# B&R Automation Studio project Nitto (part 18)

#### picctrl.ab
```automation-basic
PROGRAM _INIT
(* init program *)
wPageAct := wPageAct;
wPageOld := 255;
//wPageNew := wPageNew;
// 2012-09-11 /schoenefeldr/
wPageNew := 2;
wPageNo  := 255;

wLanguageAct := wLanguageAct;
wLanguageNew := wLanguageNew;

//-------------------------------
//access to local structures
strcpy(ADR(szPvName), "csv_hdl:CSV_Hndl");
wStatus := PV_xgetadr(ADR(szPvName),ADR(lAdrCSV_Hndl),ADR(lDataLen));
IF (wStatus = 0) THEN
	ptCSV_Hndl ACCESS lAdrCSV_Hndl;
ENDIF;

strcpy(ADR(szPvName), "tool_hdl:TOOL_Hndl");
wStatus := PV_xgetadr(ADR(szPvName),ADR(lAdrTool_Hndl),ADR(lDataLen));
IF (wStatus = 0) THEN
	ptTool_Hndl ACCESS lAdrTool_Hndl;
ENDIF;

strcpy(ADR(szPvName), "save2USB:BackupRecipes2USB");
wStatus := PV_xgetadr(ADR(szPvName),ADR(lAdrBackupRecipes2USB),ADR(lDataLen));
IF (wStatus = 0) THEN
	ptBackupRecipes2USB ACCESS lAdrBackupRecipes2USB;
ENDIF;

strcpy(ADR(szPvName), "save2USB:BackupTools2USB");
wStatus := PV_xgetadr(ADR(szPvName),ADR(lAdrBackupTools2USB),ADR(lDataLen));
IF (wStatus = 0) THEN
	ptBackupTools2USB ACCESS lAdrBackupTools2USB;
ENDIF;

strcpy(ADR(szPvName), "tool_hdl:szFileDevice");
wStatus := PV_xgetadr(ADR(szPvName),ADR(lAdrFileDeviceTool),ADR(lDataLen));
IF (wStatus = 0) THEN
	ptFileDeviceTool ACCESS lAdrFileDeviceTool;
ENDIF;

strcpy(ADR(szPvName), "tool_hdl:tmpTool");
wStatus := PV_xgetadr(ADR(szPvName),ADR(lAdrTmpTool),ADR(lDataLen));
IF (wStatus = 0) THEN
	ptTmpTool ACCESS lAdrTmpTool;
ENDIF;

	HWInfo_0.enable := TRUE;
	HWInfo_0.first := TRUE;
	HWInfo_0.pName := ADR(HWString);
	HWInfo_0 FUB HWInfo();

	AssignFirstListboxIdx		:= TRUE;
	FirstListboxIdxValid		:= FALSE;

END_PROGRAM

PROGRAM _CYCLIC
(* cyclic program *)
	TON_Cal.IN	:= (gVisu.Cmd.pageSel.actPage = 100)
	TON_Cal.PT	:= T#10s
	TON_Cal FUB TON();

	strcpy(ADR(HWString), "AR000");	//OKrebs 17.06.2014

	IF (HWString = "AR000") THEN
		IF (gVisu.Cmd.pageSel.actPage = 100) THEN
			gVisu.Cmd.pageSel.newPage := 2;
		ENDIF
	ELSE
		IF (CalibrationState = 1) AND (TON_Cal.Q) THEN
			gVisu.Cmd.pageSel.newPage := 2;
		ENDIF;
	ENDIF;

	wPageAct:=	gVisu.Cmd.pageSel.actPage

	;Blinker
TP_10ms_01.IN := NOT (TP_10ms_02.Q);
TP_10ms_01 FUB TP_10ms();
TP_10ms_02.IN := NOT (TP_10ms_01.Q);
TP_10ms_02 FUB TP_10ms();

		;-------------------------------------
;Bildwechsel erfassen
IF ((wPageAct <> wPageOld) AND (wPageNo = wPageOld)) THEN
	xPageExit := TRUE;
	wPageOld := wPageAct;
ELSE IF ((wPageNo <> wPageOld) AND (wPageNo <> wPageAct)) THEN
	xPageExit := FALSE;
	xPageInit := TRUE;
	wPageNo := wPageAct;
ELSE
	xPageInit := FALSE;
ENDIF;

;-------------------------------------
;Auswertung der Tasten in den einzelnen Bildern
CASE wPageNo OF

	ACTION P001_Recipe:				;//0,
		IF (xPageInit = TRUE) THEN
			LOOP ii := 0 TO 12 DO
			//	Button.Status[ii] := 1; //alle Tasten ausblenden
				Button.Status[ii] := 0; //alle Tasten anzeigen
			ENDLOOP;

			//strcpy(ADR(RecipeEdit.header.name), ADR(ptCSV_Hndl.FileNameSelected) );
			// 2012-12-06 /schoenefeldr/
			// Temporary solution with memcopy
			memcpy(ADR(RecipeEdit.header.name), ADR(ptCSV_Hndl.FileNameSelected), SIZEOF(RecipeEdit.header.name));
			RecipeEdit.header.name[RCP_PROG_TEXT_FILENAME_MAX] := 0;

			Button.Status[1] := 0;	//Taste anzeigen
			Button.Status[2] := 0;
			Button.Status[4] := 0;
			Button.Status[5] := 0;
			Button.Status[6] := 0;
			Button.Status[7] := 0;
			Button.Status[8] := 0;
			Button.Status[11] := 0;

				// 2013-04-18 /schoenefeldr/
				// Look for the filename in the directory and compare it to the name in the
				// Application recipe in order to restore the Listbos Index
				IF AssignFirstListboxIdx THEN
					// Search and set the index only once after warm start:
					AssignFirstListboxIdx		:= FALSE;
					// Copy the name from the recipe header into a string for comparison
					strcpy(ADR(NameFromApplRecipe), ADR(gApplRecipe.header.name) );

					// loop through the found filenames from the listbox
					LOOP ii:=0 TO USINT(ptCSV_Hndl.ListboxMaxLines) DO
						IF (strcmp(ADR(NameFromApplRecipe), ADR(ptCSV_Hndl.ListboxFileNames[ii])) = 0) THEN
							// Filename found in listbox, assign listbox index
							ptCSV_Hndl.ListboxIdx = ii;
							// Store the result, this may be evaluated later (future option)
							FirstListboxIdxValid		:= TRUE;
							// terminate loop
							EXITIF(1=1);
							ENDIF;
						ENDLOOP;
				ENDIF

		ENDIF;	//xPageInit

		//button pressed?
		IF (Button.F1 = 1) THEN
			// 2012-09-18 /schoenefeldr/
			// Immediately copy recipe data from edit recipe into application recipe
			Button.F1 := 0;
			memcpy(ADR(gApplRecipe),ADR(RecipeEdit),SIZEOF(gApplRecipe));
			// Request for updating recipe parameters
			gMachine.Command.UpdateRecipe		:= TRUE;
		ENDIF;

		IF (Button.F2 = 1) THEN
			Button.F2 := 0;
			ptCSV_Hndl.ReqDelRecipe = 1;	//start action in task csv_hdl
		ENDIF;

		IF (Button.F3 = 1) THEN
			Button.F3 := 0;
			// 2012-12-19 /schoenefeldr/
			// Copy recipe data from application recipe (actually active in the machine) into the selected recipe
			// memcpy(ADR(RecipeEdit),ADR(gApplRecipe),SIZEOF(RecipeEdit));
		ENDIF;

		IF (Button.F4 = 1) THEN
			Button.F4 := 0;
			ptCSV_Hndl.ReqNewRecipe := 1;
			ptCSV_Hndl.BtnNew := 1;
			ptCSV_Hndl.BtnSaveAs := 0;
		ENDIF;

		IF (Button.F5 = 1) THEN
			Button.F5 := 0;
			ptCSV_Hndl.ReqParaWrite := 1;
			ptCSV_Hndl.ValueChanged := 0;
		ENDIF;

		IF (Button.F6 = 1) THEN
			Button.F6 := 0;
			ptCSV_Hndl.ReqSaveAs := 1;
			ptCSV_Hndl.BtnSaveAs := 1;
			ptCSV_Hndl.BtnNew := 0;
		ENDIF;

		IF (Button.F7 = 1) THEN
			Button.F7 := 0;
			ptCSV_Hndl.ReqDirRead := 1;
		ENDIF;

		IF (Button.F8 = 1) THEN
			Button.F8 := 0;
			ptBackupRecipes2USB := TRUE;
		ENDIF;

		IF (Button.F9 = 1) THEN
			Button.F9 := 0;
		ENDIF;

		IF (Button.F10 = 1) THEN
			Button.F10 := 0;
		ENDIF;

		IF (Button.F11 = 1) THEN
			Button.F11 := 0;
			gVisu.Cmd.pageSel.newPage := P002_Tool;
		ENDIF;

		IF (Button.F12 = 1) THEN
			Button.F12 := 0;
			gVisu.Cmd.pageSel.newPage := _002_MASCHINEN_ANSICHT;
		ENDIF;

		//messagebox handling
		IF (ptCSV_Hndl.SaveFileYes = 1) THEN
			ptCSV_Hndl.SaveFileYes := 0;
			ptCSV_Hndl.ReqParaWriteAfterValueChanged := 1;
			ptCSV_Hndl.LayerMessageBoxSaveFile := 1;
		ENDIF;
		IF (ptCSV_Hndl.SaveFileNo = 1) THEN
			ptCSV_Hndl.SaveFileNo := 0;
			ptCSV_Hndl.ReqParaWriteAfterValueChanged := 0;
			ptCSV_Hndl.LayerMessageBoxSaveFile := 1;
		ENDIF;

		IF (ptCSV_Hndl.OverwriteFileYes = 1) THEN
			ptCSV_Hndl.OverwriteFileYes := 0;
			ptCSV_Hndl.FileOverWrite := 1;
			ptCSV_Hndl.LayerMessageBoxOverwrite := 1;
		ENDIF;
		IF (ptCSV_Hndl.OverwriteFileNo = 1) THEN
			ptCSV_Hndl.OverwriteFileNo := 0;
			ptCSV_Hndl.FileOverWrite := 0;
			ptCSV_Hndl.LayerMessageBoxOverwrite := 1;
		ENDIF;

		IF (ptCSV_Hndl.DeleteFileYes = 1) THEN
			ptCSV_Hndl.DeleteFileYes := 0;
			ptCSV_Hndl.FileDelete = 1;
			ptCSV_Hndl.LayerMessageBoxDeleteFile := 1;
		ENDIF;
		IF (ptCSV_Hndl.DeleteFileNo = 1) THEN
			ptCSV_Hndl.DeleteFileNo := 0;
			ptCSV_Hndl.FileDelete = 0;
			ptCSV_Hndl.LayerMessageBoxDeleteFile := 1;
		ENDIF;

		//---------------------------------
		//was another recipe selected in list ?
		IF (ptCSV_Hndl.ListBoxRecipeChanged = TRUE) THEN
			//strcpy(ADR(RecipeEdit.header.name), ADR(ptCSV_Hndl.FileNameSelected) );
			// 2012-12-06 /schoenefeldr/
			// Temporary solution with memcopy
			memcpy(ADR(RecipeEdit.header.name), ADR(ptCSV_Hndl.FileNameSelected), SIZEOF(RecipeEdit.header.name));
			RecipeEdit.header.name[RCP_PROG_TEXT_FILENAME_MAX] := 0;
			ptCSV_Hndl.ListBoxRecipeChanged := FALSE;

			ptCSV_Hndl.StatusBmpFoundFileCutU1 = VISIBLE;	//show bmp
			ptCSV_Hndl.StatusBtnRefreshCutU1 := INVISIBLE;	//but don't show text and button
			LOOP ii:=0 TO USINT(ptTool_Hndl.ListboxMaxLines) DO
				IF (strcmp(ADR(RecipeEdit.cutUnit1.toolfilename), ADR(ptTool_Hndl.ListboxFileNames[ii])) = 0) THEN
					RecipeEdit.cutUnit1.toolNumber = ii;
					ptCSV_Hndl.StatusBmpFoundFileCutU1 = INVISIBLE;	//don't show bmp
					ptCSV_Hndl.StatusBtnRefreshCutU1 := VISIBLE;	//but show text and button
					EXITIF(1=1);
				ENDIF;
			ENDLOOP;

			ptCSV_Hndl.StatusBmpFoundFileCutU2 = VISIBLE;	//show bmp
			ptCSV_Hndl.StatusBtnRefreshCutU2 := INVISIBLE;	//but don't show text and button
			LOOP ii:=0 TO USINT(ptTool_Hndl.ListboxMaxLines) DO
				IF (strcmp(ADR(RecipeEdit.cutUnit2.toolfilename), ADR(ptTool_Hndl.ListboxFileNames[ii])) = 0) THEN
					RecipeEdit.cutUnit2.toolNumber = ii;
					ptCSV_Hndl.StatusBmpFoundFileCutU2 := INVISIBLE;	//don't show bmp
					ptCSV_Hndl.StatusBtnRefreshCutU2 := VISIBLE;	//but show text and button
					EXITIF(1=1);
				ENDIF;
			ENDLOOP;

;			ptCSV_Hndl.StatusBmpFoundFileCutU3 = VISIBLE;	//show bmp
;			ptCSV_Hndl.StatusBtnRefreshCutU3 := INVISIBLE;	//but don't show text and button
;			LOOP ii:=0 TO USINT(ptTool_Hndl.ListboxMaxLines) DO
;				IF (strcmp(ADR(RecipeEdit.cutUnit3.toolfilename), ADR(ptTool_Hndl.ListboxFileNames[ii])) = 0) THEN
;					RecipeEdit.cutUnit3.toolNumber = ii;
;					ptCSV_Hndl.StatusBmpFoundFileCutU3 := INVISIBLE;	//don't show bmp
;					ptCSV_Hndl.StatusBtnRefreshCutU3 := VISIBLE;	//but show text and button
;					EXITIF(1=1);
;				ENDIF;
;			ENDLOOP;

		ENDIF;

		//---------------------------------
		//tool file was changed in cut unit 1
		IF (ptCSV_Hndl.ToolSelectedCutU1 = TRUE) THEN
			ptCSV_Hndl.ToolSelectedCutU1 := FALSE;
			ptCSV_Hndl.ValueChanged := TRUE;
			strcpy(ADR(RecipeEdit.cutUnit1.toolfilename), ADR(ptTool_Hndl.ListboxFileNames[RecipeEdit.cutUnit1.toolNumber]));
			strcpy(ADR(szToolFileName), ADR(RecipeEdit.cutUnit1.toolfilename));
			lAdrDestination := ADR(RecipeEdit.cutUnit1.tool);  //where to copy the data
			xReadToolFile := TRUE;
		ENDIF;

		//---------------------------------
		//tool file was changed in cut unit 2
		IF (ptCSV_Hndl.ToolSelectedCutU2 = TRUE) THEN
			ptCSV_Hndl.ToolSelectedCutU2 := FALSE;
			ptCSV_Hndl.ValueChanged := TRUE;
			strcpy(ADR(RecipeEdit.cutUnit2.toolfilename), ADR(ptTool_Hndl.ListboxFileNames[RecipeEdit.cutUnit2.toolNumber]));
			strcpy(ADR(szToolFileName), ADR(RecipeEdit.cutUnit2.toolfilename));
			lAdrDestination := ADR(RecipeEdit.cutUnit2.tool);   //where to copy the data
			xReadToolFile := TRUE;
		ENDIF;

		//---------------------------------
		//tool file was changed in cut unit 3
		IF (ptCSV_Hndl.ToolSelectedCutU3 = TRUE) THEN
			ptCSV_Hndl.ToolSelectedCutU3 := FALSE;
			ptCSV_Hndl.ValueChanged := TRUE;
			strcpy(ADR(RecipeEdit.cutUnit3.toolfilename), ADR(ptTool_Hndl.ListboxFileNames[RecipeEdit.cutUnit3.toolNumber]));
			strcpy(ADR(szToolFileName), ADR(RecipeEdit.cutUnit3.toolfilename));
			lAdrDestination := ADR(RecipeEdit.cutUnit3.tool);   //where to copy the data
			xReadToolFile := TRUE;
		ENDIF;
		//---------------------------------

		IF (xPageExit = TRUE) THEN

		ENDIF;

	ENDACTION;

	;-----------------------------------
	ACTION P002_Tool:				;//1,
		IF (xPageInit = TRUE) THEN
			LOOP ii := 0 TO 12 DO
//				Button.Status[ii] := 1; //alle Tasten ausblenden
				Button.Status[ii] := 0; //alle Tasten anzeigen
			ENDLOOP;
			Button.Status[2] := 0;	//Taste anzeigen
			Button.Status[4] := 0;
			Button.Status[5] := 0;
			Button.Status[6] := 0;
			Button.Status[7] := 0;
			Button.Status[8] := 0;
			Button.Status[11] := 0;
		ENDIF;

		//button pressed?
		IF (Button.F1 = 1) THEN
			Button.F1 := 0;
		ENDIF;

		IF (Button.F2 = 1) THEN
			Button.F2 := 0;
			ptTool_Hndl.ReqDelRecipe = 1;	//start action in task csv_hdl
		ENDIF;

		IF (Button.F3 = 1) THEN
			Button.F3 := 0;
		ENDIF;

		IF (Button.F4 = 1) THEN
			Button.F4 := 0;
			ptTool_Hndl.ReqNewRecipe := 1;
			ptTool_Hndl.BtnNew := 1;
			ptTool_Hndl.BtnSaveAs := 0;
		ENDIF;

		IF (Button.F5 = 1) THEN
			Button.F5 := 0;
			ptTool_Hndl.ReqParaWrite := 1;
			ptTool_Hndl.ValueChanged := 0;
		ENDIF;

		IF (Button.F6 = 1) THEN
			Button.F6 := 0;
			ptTool_Hndl.ReqSaveAs := 1;
			ptTool_Hndl.BtnSaveAs := 1;
			ptTool_Hndl.BtnNew := 0;
		ENDIF;

		IF (Button.F7 = 1) THEN
			Button.F7 := 0;
			ptTool_Hndl.ReqDirRead := 1;
		ENDIF;

		IF (Button.F8 = 1) THEN
			Button.F8 := 0;
			ptBackupTools2USB := TRUE;
		ENDIF;

		IF (Button.F9 = 1) THEN
			Button.F9 := 0;
		ENDIF;

		IF (Button.F10 = 1) THEN
			Button.F10 := 0;
		ENDIF;

		IF (Button.F11 = 1) THEN
			Button.F11 := 0;
		ENDIF;

		IF (Button.F12 = 1) THEN
			Button.F12 := 0;
			gVisu.Cmd.pageSel.newPage := _002_MASCHINEN_ANSICHT;
		ENDIF;

		//messagebox handling
		IF (ptTool_Hndl.SaveFileYes = 1) THEN
			ptTool_Hndl.SaveFileYes := 0;
			ptTool_Hndl.ReqParaWriteAfterValueChanged := 1;
			ptTool_Hndl.LayerMessageBoxSaveFile := 1;
		ENDIF;
		IF (ptTool_Hndl.SaveFileNo = 1) THEN
			ptTool_Hndl.SaveFileNo := 0;
			ptTool_Hndl.ReqParaWriteAfterValueChanged := 0;
			ptTool_Hndl.LayerMessageBoxSaveFile := 1;
		ENDIF;

		IF (ptTool_Hndl.OverwriteFileYes = 1) THEN
			ptTool_Hndl.OverwriteFileYes := 0;
			ptTool_Hndl.FileOverWrite := 1;
			ptTool_Hndl.LayerMessageBoxOverwrite := 1;
		ENDIF;
		IF (ptTool_Hndl.OverwriteFileNo = 1) THEN
			ptTool_Hndl.OverwriteFileNo := 0;
			ptTool_Hndl.FileOverWrite := 0;
			ptTool_Hndl.LayerMessageBoxOverwrite := 1;
		ENDIF;

		IF (ptTool_Hndl.DeleteFileYes = 1) THEN
			ptTool_Hndl.DeleteFileYes := 0;
			ptTool_Hndl.FileDelete = 1;
			ptTool_Hndl.LayerMessageBoxDeleteFile := 1;
		ENDIF;
		IF (ptTool_Hndl.DeleteFileNo = 1) THEN
			ptTool_Hndl.DeleteFileNo := 0;
			ptTool_Hndl.FileDelete = 0;
			ptTool_Hndl.LayerMessageBoxDeleteFile := 1;
		ENDIF;

		IF (xPageExit = TRUE) THEN

		ENDIF;
	ENDACTION;

	;-----------------------------------
	ACTION P003_AlarmCurrent:				;//2,
		if (xPageInit = TRUE) then
			LOOP ii := 0 TO 12 DO
//				Button.Status[ii] := 1; //alle Tasten ausblenden
				Button.Status[ii] := 0; //alle Tasten anzeigen
			ENDLOOP;

			Button.Status[11] := 0;	//Taste anzeigen
		ENDIF;

		//button pressed?
		IF (Button.F1 = 1) THEN
			Button.F1 := 0;
		ENDIF;

		IF (Button.F2 = 1) THEN
			Button.F2 := 0;
		ENDIF;

		IF (Button.F3 = 1) THEN
			Button.F3 := 0;
		ENDIF;

		IF (Button.F4 = 1) THEN
			Button.F4 := 0;
		ENDIF;

		IF (Button.F5 = 1) THEN
			Button.F5 := 0;
		ENDIF;

		IF (Button.F6 = 1) THEN
			Button.F6 := 0;
		ENDIF;

		IF (Button.F7 = 1) THEN
			Button.F7 := 0;
		ENDIF;

		IF (Button.F8 = 1) THEN
			Button.F8 := 0;
		ENDIF;

		IF (Button.F9 = 1) THEN
			Button.F9 := 0;
		ENDIF;

		IF (Button.F10 = 1) THEN
			Button.F10 := 0;
		ENDIF;

		IF (Button.F11 = 1) THEN
			Button.F11 := 0;
		ENDIF;

		IF (Button.F12 = 1) THEN
			Button.F12 := 0;
			gVisu.Cmd.pageSel.newPage := _002_MASCHINEN_ANSICHT;
		ENDIF;

		IF (xPageExit = TRUE) THEN

		ENDIF;
	ENDACTION;

	;-----------------------------------
	ACTION P004_AlarmHistory:			;//3
		IF (xPageInit = TRUE) THEN

		ENDIF;

		IF (xPageExit = TRUE) THEN

		ENDIF;
	ENDACTION;

ENDCASE;	//of wPageNr

CASE bStepCmd OF
	ACTION ST_WAIT:
		IF (xReadToolFile = TRUE) THEN
			xReadToolFile := FALSE;
			bStepCmd := READ_TOOL_FILE;
		ENDIF;
	ENDACTION;

	ACTION READ_TOOL_FILE:
		CSV_ReadToolFile.pFileName := ADR(szToolFileName);	//ADR(RecipeEdit.cutUnit1.toolfilename);
		CSV_ReadToolFile.pDevice :=  ADR(ptFileDeviceTool);	//  "DIR_TOOL";
		CSV_ReadToolFile.No_DatatypControl := 1;
		CSV_ReadToolFile.Separator := 59;
		CSV_ReadToolFile.IgnoreError := 1;

		CSV_ReadToolFile FUB CSV_ReadFile();

		retval := CSV_ReadToolFile.status;
		IF (retval = 0) THEN
			//after reading the file, the values are in 'tool_hdl:tmpTool'
			memcpy(lAdrDestination, ADR(ptTmpTool), SIZEOF(ptTmpTool));
			bStepCmd := ST_WAIT;
		ELSE IF (retval = ERR_FUB_BUSY) THEN
			;
		ELSE
			bStepCmd := ST_WAIT;
		ENDIF;
	ENDACTION;
		ENDCASE;	//of bStepCmd

END_PROGRAM
```

#### picctrl.var
```iecst
VAR
	bStepCmd : USINT;
	CSV_ReadToolFile : CSV_ReadFile;
	ii : USINT;
END_VAR
VAR CONSTANT
	INVISIBLE : USINT := 1;
END_VAR
VAR
	lAdrBackupRecipes2USB : UDINT;
	lAdrBackupTools2USB : UDINT;
	lAdrCSV_Hndl : UDINT;
	lAdrDestination : UDINT;
	lAdrFileDeviceTool : UDINT;
	lAdrTmpTool : UDINT;
	lAdrTool_Hndl : UDINT;
	lDataLen : UDINT;
END_VAR
VAR CONSTANT
	P001_Recipe : UINT := 110;
	P002_Tool : UINT := 111;
	P003_AlarmCurrent : UINT := 112;
	P004_AlarmHistory : UINT := 113;
	_002_MASCHINEN_ANSICHT : UINT := 2;
END_VAR
VAR
	ptBackupRecipes2USB : REFERENCE TO BOOL;
	ptBackupTools2USB : REFERENCE TO BOOL;
	ptCSV_Hndl : REFERENCE TO CSVHndl_typ;
	ptFileDeviceTool : REFERENCE TO STRING[80];
	ptTmpTool : REFERENCE TO rcp_tool_typ;
	ptTool_Hndl : REFERENCE TO TOOL_Hndl_typ;
END_VAR
VAR CONSTANT
	READ_TOOL_FILE : USINT := 5;
END_VAR
VAR
	retval : UINT;
	szPvName : STRING[80];
	szToolFileName : STRING[80];
	TP_10ms_01 : TP_10ms;
	TP_10ms_02 : TP_10ms;
END_VAR
VAR CONSTANT
	VISIBLE : USINT := 0;
	ST_WAIT : USINT := 0;
END_VAR
VAR
	wLanguageAct : UINT;
	wLanguageNew : UINT;
	wPageAct : UINT;
	wPageNew : UINT;
	wPageNo : UINT;
	wPageOld : UINT;
	wStatus : UINT;
	xPageExit : BOOL;
	xPageInit : BOOL;
	xReadToolFile : BOOL;
	CalibrationState : INT;
	TON_Cal : TON;
	HWString : STRING[20] := 'AR000';
END_VAR
(*Restore list box index after warmstart*)
VAR
	AssignFirstListboxIdx : BOOL; (*Flag for restoring the index only once*)
	FirstListboxIdxValid : BOOL; (*Flag for found filename (optional evaluation, future use)*)
	NameFromApplRecipe : STRING[80]; (*local filename, converted from application recipe header*)
	HWInfo_0 : HWInfo;
END_VAR
```

### Package Logical/Alarme - Alarme erzeugen für alle BG

### Program Logical/Alarme/GeneralAlarms (IEC) - Ein neues Programm

#### GeneralAlarms.st - Implementierungscode
```iecst
(********************************************************************
 * COPYRIGHT --
 ********************************************************************
 * Programm: GeneralAlarms
 * Datei: GeneralAlarms.st
 * Autor: jkappelt
 * Erstellt: 3. Oktober 2012
 ********************************************************************
 * Implementierung des Programms GeneralAlarms
 ********************************************************************)

PROGRAM _INIT

(* TODO : Code hier einfügen *)

END_PROGRAM

PROGRAM _CYCLIC
// Reset Alarme
	IF gMachine.IO.DIn.LDT_FaultReset.Value.InVal THEN
		gMachine.Command.AutoStopRequestAlarm := FALSE;	//reset stop request
		FOR i := 0 TO 23 BY 1 DO
			GeneralAlarm[i] := 0;
			AlarmWinder[i]	:= 0;
		END_FOR;
	END_IF;

//
//	IF 	NOT	gMachine.IO.DIn.PressureCtrl.Value.InVal AND gMachine.IO.DIn.LDT_Reset.Value.State AND  AxisIf.Status.drivesEnabled THEN
//		GeneralAlarm[ALARM_PRESSURE_LOW] := TRUE;
//	END_IF;
	GeneralAlarm[ALARM_FUSE_BST] :=	NOT	gMachine.IO.DIn.FuseBTS.Value.InVal;
	GeneralAlarm[ALARM_FUSE_QW258] :=	NOT	gMachine.IO.DIn.FuseQW258_262.Value.InVal;
//	GeneralAlarm[3] :=	NOT	gMachine.IO.DIn.FuseQW264_268.Value.InVal;
	// GeneralAlarm[4]:= siehe unten
	GeneralAlarm[ALARM_ESTOP_CABINET] := NOT gMachine.IO.DIn.EmergencyStopCabinet.Value.InVal;
	GeneralAlarm[ALARM_ESTOP_PANEL] := NOT gMachine.IO.DIn.EmergencyStopPanel.Value.InVal;
	GeneralAlarm[ALARM_ESTOP_UNWINDER] := NOT gMachine.IO.DIn.EmergencyStopUnwinder.Value.InVal;
	GeneralAlarm[ALARM_ESTOP_MIDDLE] := NOT gMachine.IO.DIn.EmergencyStopMiddle.Value.InVal;
	GeneralAlarm[ALARM_ESTOP_ENDMODULE] := NOT gMachine.IO.DIn.EmergencyStopEndModule.Value.InVal;
	GeneralAlarm[ALARM_ESTOP_BOOKLET] := NOT gMachine.IO.DIn.EmergencyStopBooklet.Value.InVal;

	//	GeneralAlarm[9] := NOT	gMachine.IO.DIn.EmergencyStopTandemWinder.Value.InVal;

//	GeneralAlarm[ALARM_FUSE_COOLER_UNWINDER] :=	NOT	gMachine.IO.DIn.FuseFanUnwind.Value.InVal ;

	GeneralAlarm[ALARM_PLUG1] :=	NOT	gMachine.IO.DIn.FusePlug1.Value.InVal;
	GeneralAlarm[ALARM_PLUG2] :=	NOT	gMachine.IO.DIn.FusePlug2.Value.InVal;
	GeneralAlarm[ALARM_PLUGCEE] :=	NOT	gMachine.IO.DIn.FusePlugCEE.Value.InVal;
	GeneralAlarm[ALARM_FUSE_BOOKLET] :=	NOT	gMachine.IO.DIn.FuseBookletFeeder.Value.InVal;
	GeneralAlarm[ALARM_SAFEDOOR_BOOKLET] :=	NOT	gMachine.IO.DIn.SafetyDoorBooklet.Value.InVal AND gMachine.IO.DIn.EmergencyStopBooklet.Value.InVal;
	GeneralAlarm[ALARM_ESTOP_PULLWIRE] :=	NOT	gMachine.IO.DIn.EmergencyStopPullWire.Value.InVal;

	//	GeneralAlarm[ALARM_HVOLT_ANTISTATIC] :=	NOT	gMachine.IO.DIn.HighVoltageGenerator.Value.InVal;

//	GeneralAlarm[ALARM_BST_NREADY] 		:= NOT	gMachine.IO.DIn.BST_OK.Value.InVal;
	GeneralAlarm[ALARM_SAFEDOOR_PUNCH1] := NOT gMachine.IO.DIn.SafetyDoorInfeedCut1.Value.InVal OR NOT gMachine.IO.DIn.SafetyDoorOutfeedCut1.Value.InVal;
	GeneralAlarm[ALARM_SAFEDOOR_PUNCH2] := NOT gMachine.IO.DIn.SafetyDoorInfeedCut2.Value.InVal OR NOT gMachine.IO.DIn.SafetyDoorOutfeedCut2.Value.InVal;
//	GeneralAlarm[ALARM_SAFEDOOR_PUNCH3] := NOT gMachine.IO.DIn.SafetyDoorInfeedCut3.Value.InVal OR NOT gMachine.IO.DIn.SafetyDoorOutfeedCut3.Value.InVal;
	GeneralAlarm[ALARM_SAFEDOOR_LONGCUT]:= NOT gMachine.IO.DIn.SafetyDoorLongCut.Value.InVal;
//	GeneralAlarm[ALARM_FUSE_LAMINATOR]	:= NOT gMachine.IO.DIn.Fuse_Laminator.Value.InVal;
	GeneralAlarm[ALARM_WEB_BREAK]		:= gMachine.Status.WebBreakLabeler;

	Speed_machine := REAL_TO_INT(gVisu.Status.ActVelocity /1000);

	IF Speed_machine <= 1 THEN
		Machine_Stop := 0;
	ELSE
		Machine_Stop := 1;
	END_IF;

	//reset Button am Panel Setz Fehler nummer zurück

	IF gMachine.IO.DIn.LDT_FaultReset.Value.InVal THEN
		IF gMachine.IO.DIn.LDT_FaultReset.Value.InVal THEN
			AlarmUnwinder[1]:=0;
			AlarmEndModul[4] := 0;
			AlarmEndModul[5] := 0;
			GeneralAlarm[4] := 0;
		END_IF ;

	END_IF;
	//********************	Safety Status auf Panel anzeigen  *********************************************************
	IF (gMachine.Safety.RequestSTO) THEN
		StatusSafety	:=	STATUS_CONTVOL_OFF;
	ELSIF (gMachine.Safety.RequestSLS) THEN
		StatusSafety	:=	STATUS_SLS;
	ELSE
		StatusSafety	:=	STATUS_SAFETY_OK;
	END_IF;
	//******************************************************************************************************************

	//********************	Stop-Anforderung durch Unterschreitung des min. Durchmessers Unwinder!!	********************
	TON_LowDiamUnwinder.PT	:= T#2s;
	TON_LowDiamUnwinder.IN	:= (gMachine.Status.CalcDiam.MainUnwind < gMachRecipe.mainUnwind.StopDiam) AND gMachine.Status.mAutoModeActive AND gApplRecipe.dancer.radiusCtrlOn;
	TON_LowDiamUnwinder();

	IF 	(TON_LowDiamUnwinder.Q) THEN
		gMachine.Command.AutoStopRequestAlarm := TRUE;
		AlarmUnwinder[1]:=1;
	END_IF;
	//****************************************************************************************************

	//** Splicetable Unwinder ******************************************************)
	IF gMachine.IO.DOut.VentCutTabOutfeedMoveUpDn.Value.State OR gMachine.IO.DOut.VentCutTabInfeedMoveUpDn.Value.State THEN
		AlarmUnwinder[5]:= TRUE;
	END_IF

	//********************	Stop-Anforderung durch Überschreitung des max. Durchmessers Tandemwickler!!	********************
//	TON_HighDiamTWindTop.PT	:= T#3s;
//	TON_HighDiamTWindTop.IN	:= (gMachine.Status.Diam.TUnwindTop > gMachRecipe.topTandemWind.StopDiam) AND AxisIf.Status.isMoving;
//	TON_HighDiamTWindTop();
//
//	IF (TON_HighDiamTWindTop.Q) THEN
//		gMachine.Command.AutoStopRequestAlarm := TRUE;
//		AlarmEndModul[4] := 1;
//	END_IF;
//
//	TON_HighDiamTWindBot.PT	:= T#3s;
//	TON_HighDiamTWindBot.IN	:= (gMachine.Status.Diam.TUnwindBot > gMachRecipe.botTandemWind.StopDiam) AND AxisIf.Status.isMoving;
//	TON_HighDiamTWindBot();
//
//	IF 	(TON_HighDiamTWindBot.Q) THEN
//		gMachine.Command.AutoStopRequestAlarm := TRUE;
//		AlarmEndModul[5] := 1;
//	END_IF;
	//****************************************************************************************************

	//********************	Stop-Anforderung der Aufwickler und Abwickler!!	********************

	// Spender //
	// Stop-Anforderung durch Überschreitung des min. Durchmessers Aufwickler!!
	IF 	gMachine.Status.Diam.Spend1	 > gMachRecipe.spender1.StopDiam AND (gApplRecipe.spender1.mode = 1)  THEN
		gMachine.Command.AutoStopRequestAlarm := TRUE;
		AlarmWinder[0] := 1;
	END_IF;
	// Stop-Anforderung durch Unterschreitung des min. Durchmessers Abwickler!!
	IF 	gMachine.Status.Diam.Spend2 < gMachRecipe.spender2.StopDiam  AND  (gApplRecipe.spender1.mode = 1) THEN
		gMachine.Command.AutoStopRequestAlarm := TRUE;
		AlarmWinder[1] := 1;
	END_IF;

	// Laminierer //
	// Stop-Anforderung durch Unterschreitung des min. Durchmessers Abwickler!!
	IF 	gMachine.Status.Diam.Laminator1 < gMachRecipe.laminator1.StopDiam  AND (gApplRecipe.laminator2.mode = 36 )  THEN
		gMachine.Command.AutoStopRequestAlarm := TRUE;
		AlarmWinder[2] := 1;
	END_IF;
	// Stop-Anforderung durch Überschreitung des min. Durchmessers Aufwickler!!
	IF 	gMachine.Status.Diam.Laminator2	 > gMachRecipe.laminator2.StopDiam AND (gApplRecipe.laminator2.mode = 36 )  THEN
		gMachine.Command.AutoStopRequestAlarm := TRUE;
		AlarmWinder[3] := 1;
	END_IF;

	// Gitteraufwickler 1 //
	// Stop-Anforderung durch Überschreitung des min. Durchmessers Aufwickler!!
	IF 	gMachine.Status.Diam.Grid1	 > gMachRecipe.grid1.StopDiam AND (gApplRecipe.grid1.mode = 36)  THEN
		gMachine.Command.AutoStopRequestAlarm := TRUE;
		AlarmWinder[4] := 1;
	END_IF;
	// Gitteraufwickler 2 //
	// Stop-Anforderung durch Überschreitung des min. Durchmessers Aufwickler!!
	IF 	gMachine.Status.Diam.Grid2	 > gMachRecipe.grid2.StopDiam AND (gApplRecipe.grid2.mode = 36)  THEN
		gMachine.Command.AutoStopRequestAlarm := TRUE;
		AlarmWinder[5] := 1;
	END_IF;
	//****************************************************************************************************

	//********************	Stop-Anforderung durch Unterschreitung der Bahnspannung!!	********************
//	TON_LowTension.PT	:= T#1s;
//	TON_LowTension.IN	:=
//	(gMachine.IO.AIn.FlengeDMS.Value.Scaled < 5.0)
//	AND gMachine.Status.mAutoModeActive
//	AND AxisHandle[AXIS_PULL_BRAKE_ST1].Data.config.IS_ACTIVE;

	TON_LowTension();

	IF (TON_LowTension.Q) THEN
		gMachine.Command.AutoStopRequestAlarm := TRUE;
		GeneralAlarm[4] := 1;
	END_IF;
	//****************************************************************************************************

	//********************	Stop-Anforderung durch Bahnriss am Spender!!	********************
	IF (gMachine.Status.WebBreakLabeler) THEN
		gMachine.Command.AutoStopRequestAlarm := TRUE;
		GeneralAlarm[21] := 1;
	END_IF;
	//****************************************************************************************************

	// Warnung Regelung der Abwicklung nicht aktiv
	IF (gApplRecipe.mainUnwind.mode = 0) THEN
		AlarmUnwinder[11]:=1;
	END_IF
	//*******************************************************************************************************

	// Erzeugung der Vorwarnungen für min. und max. Diameter

	// Reset Warnmeldungen
	IF gMachine.IO.DIn.LDT_FaultReset.Value.InVal THEN
		AlarmUnwinder[10]:=0;
		AlarmUnwinder[11]:=0;

		AlarmEndModul[10] := 0;
		AlarmEndModul[11] := 0;
	END_IF ;
	// Warnnung max. Durchmessers!!
	IF 	(gMachine.Status.CalcDiam.MainUnwind < gMachRecipe.mainUnwind.WarnDiam) AND gMachine.Status.mAutoModeActive
		AND gApplRecipe.dancer.radiusCtrlOn THEN
		AlarmUnwinder[10]:=1;
	END_IF;

//	// Warnnung max. Durchmessers!!
//	IF 	(gMachine.Status.Diam.TUnwindTop	 > gMachRecipe.topTandemWind.WarnDiam) AND  AxisIf.Status.isMoving AND
//		((gApplRecipe.endModule.mode = 41) OR (gApplRecipe.endModule.mode = 43)) THEN
//		AlarmEndModul[10] := 1;
//	END_IF;
//	// Warnnung max. Durchmessers!!
//	IF 	(gMachine.Status.Diam.TUnwindBot> gMachRecipe.botTandemWind.WarnDiam) AND  AxisIf.Status.isMoving AND
//		((gApplRecipe.endModule.mode = 42) OR (gApplRecipe.endModule.mode = 43)) THEN
//		AlarmEndModul[11] := 1;
//	END_IF;
//

END_PROGRAM
```

#### GeneralAlarms.typ - Lokale Datentypen
```iecst
(********************************************************************
 * COPYRIGHT --
 ********************************************************************
 * Programm: GeneralAlarms
 * Datei: GeneralAlarms.typ
 * Autor: jkappelt
 * Erstellt: 3. Oktober 2012
 ********************************************************************
 * Lokale Datentypen des Programs GeneralAlarms
 ********************************************************************)

TYPE
	emuAlarmsGeneral :
		(
		ALARM_PRESSURE_LOW := 0,
		ALARM_FUSE_BST := 1,
		ALARM_FUSE_QW258 := 2,
		ALARM_FUSE_QW264 := 3,
		ALARM_LOW_WEBTENSION := 4,
		ALARM_ESTOP_CABINET := 5,
		ALARM_ESTOP_PANEL := 6,
		ALARM_ESTOP_UNWINDER := 7,
		ALARM_ESTOP_MIDDLE := 8,
		ALARM_ESTOP_ENDMODULE := 9,
		ALARM_FUSE_COOLER_UNWINDER := 10,
		ALARM_PLUG1 := 11,
		ALARM_PLUG2 := 12,
		ALARM_PLUGCEE := 13,
		ALARM_HVOLT_ANTISTATIC := 14,
		ALARM_BST_NREADY := 15,
		ALARM_SAFEDOOR_PUNCH1 := 16,
		ALARM_SAFEDOOR_PUNCH2 := 17,
		ALARM_SAFEDOOR_PUNCH3 := 18,
		ALARM_SAFEDOOR_LONGCUT := 19,
		ALARM_FUSE_LAMINATOR := 20,
		ALARM_WEB_BREAK := 21,
		ALARM_ESTOP_BOOKLET := 22,
		ALARM_FUSE_BOOKLET := 23,
		ALARM_SAFEDOOR_BOOKLET := 24,
		ALARM_ESTOP_PULLWIRE := 25
		);
	emuSafetyStatus :
		(
		STATUS_SAFETY_OK := 0,
		STATUS_SLS := 1,
		STATUS_CONTVOL_OFF := 2
		);
END_TYPE
```

#### GeneralAlarms.var - Lokale Variablen
```iecst
(********************************************************************
 * COPYRIGHT --
 ********************************************************************
 * Programm: GeneralAlarms
 * Datei: GeneralAlarms.var
 * Autor: jkappelt
 * Erstellt: 3. Oktober 2012
 ********************************************************************
 * Lokale Variablen des Programms GeneralAlarms
 ********************************************************************)
VAR
	i : SINT;
	GeneralAlarm : ARRAY[0..29] OF BOOL;
	AlarmEndModul : ARRAY[0..19] OF BOOL := [20(FALSE)];
	AlarmGridWinder : ARRAY[0..19] OF BOOL := [20(FALSE)];
	AlarmSpender : ARRAY[0..19] OF BOOL := [20(FALSE)];
	AlarmWinder : ARRAY[0..19] OF BOOL := [20(FALSE)];
	AlarmUnwinder : ARRAY[0..19] OF BOOL := [20(FALSE)];
	StatusSafety : emuSafetyStatus;
	Speed_machine : INT;
	Machine_Stop : BOOL;
	TON_LowTension : TON; (*timeout when material tension is too low*)
	TON_HighDiamTWindBot : TON; (*timeout when diameter is too high*)
	TON_HighDiamTWindTop : TON; (*timeout when diameter is too high*)
	TON_LowDiamUnwinder : TON; (*timeout when diameter is too low*)
END_VAR
```
